//{{V2}}
ORGANIZATION_BLOCK OB1
TITLE= "Cyclic main program"


AUTHOR:nb
FAMILY:nb
NAME:nb
VERSION:1.0


VAR_TEMP
       OB1_EV_CLASS:BYTE //Bits 0-3 = 1 (Coming event), Bits 4-7 = 1 (Event class 1)
       OB1_SCAN_1:BYTE //1 (Cold restart scan 1 of OB 1), 3 (Scan 2-n of OB 1)
       OB1_PRIORITY:BYTE //1 (Priority of 1 is lowest)
       OB1_OB_NUMBR:BYTE //1 (Organization block 1, OB1)
       OB1_RESERVED_1:BYTE //Reserved for system
       OB1_RESERVED_2:BYTE //Reserved for system
       OB1_PREV_CYCLE:INT //Cycle time of previous OB1 scan (milliseconds)
       OB1_MIN_CYCLE:INT //Minimum cycle time of OB1 (milliseconds)
       OB1_MAX_CYCLE:INT //Maximum cycle time of OB1 (milliseconds)
       OB1_DATE_TIME:DATE_AND_TIME //Date and time OB1 started
END_VAR
BEGIN

NETWORK
TITLE=
//{{k}}
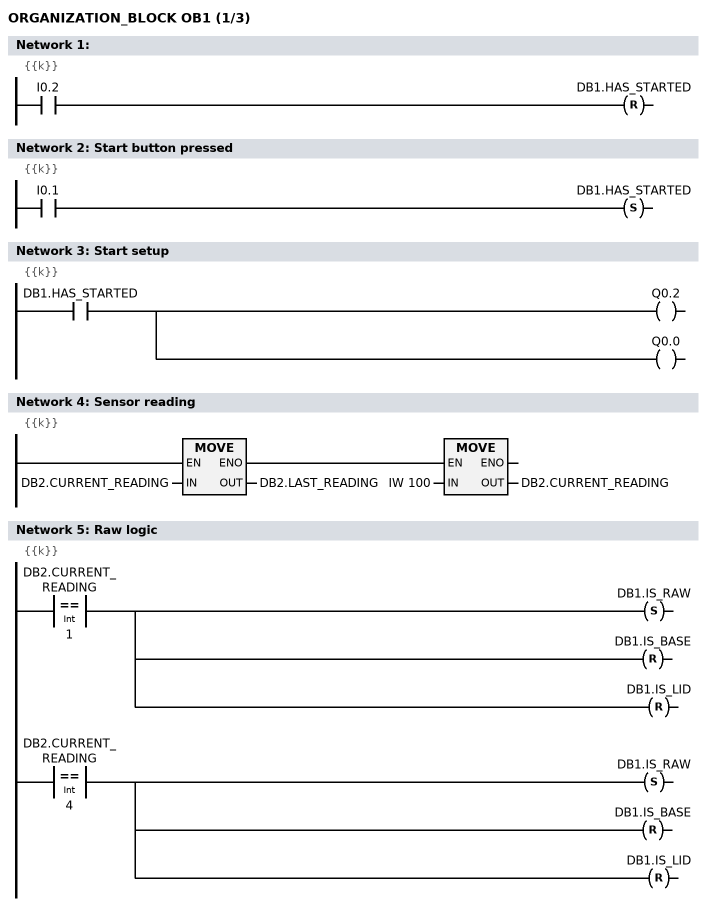

       A    I0.2
       R    DB1.HAS_STARTED

NETWORK
TITLE=Start button pressed
//{{k}}

       A    I0.1
       S    DB1.HAS_STARTED

NETWORK
TITLE=Start setup
//{{k}}

       A    DB1.HAS_STARTED
       =    Q0.2
       =    Q0.0

NETWORK
TITLE=Sensor reading
//{{k}}

       L    DB2.CURRENT_READING
       T    DB2.LAST_READING
       SET
       SAVE
       CLR
       A    BR
       JNB  _001
       L    IW        100
       T    DB2.CURRENT_READING
_001  :NOP  0
NETWORK
TITLE=Raw logic
//{{k}}

       A(
       L    DB2.CURRENT_READING
       L    1
       ==I
       )
       S    DB1.IS_RAW
       R    DB1.IS_BASE
       R    DB1.IS_LID
       A(
       L    DB2.CURRENT_READING
       L    4
       ==I
       )
       S    DB1.IS_RAW
       R    DB1.IS_BASE
       R    DB1.IS_LID
NETWORK
TITLE=Raw logic
//{{k}}
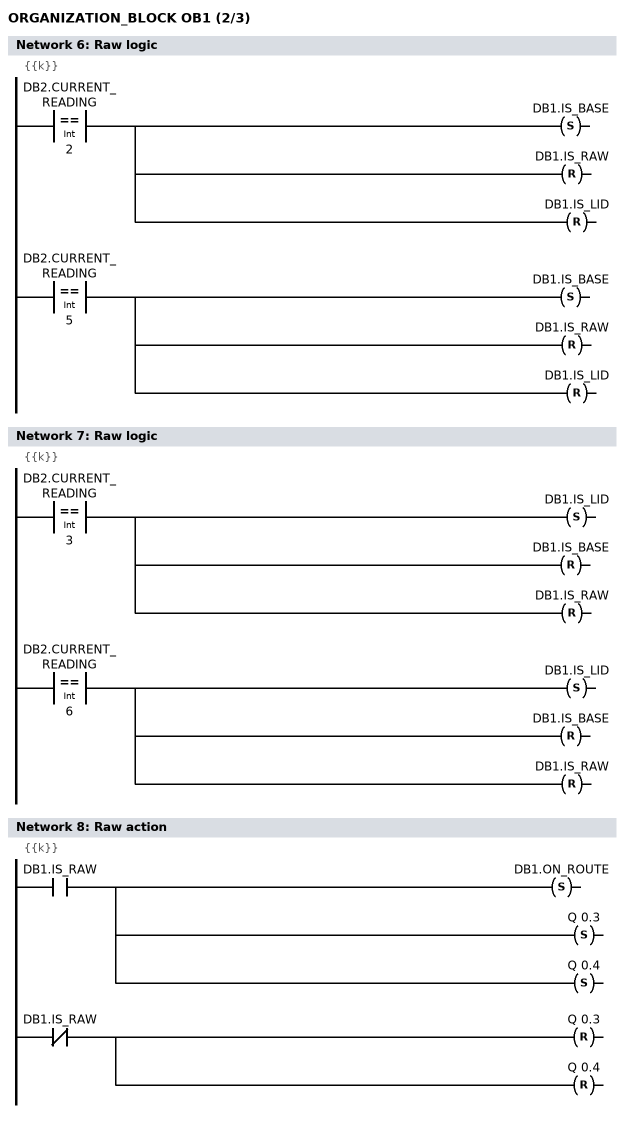

       A(
       L    DB2.CURRENT_READING
       L    2
       ==I
       )
       S    DB1.IS_BASE
       R    DB1.IS_RAW
       R    DB1.IS_LID
       A(
       L    DB2.CURRENT_READING
       L    5
       ==I
       )
       S    DB1.IS_BASE
       R    DB1.IS_RAW

       R    DB1.IS_LID
NETWORK
TITLE=Raw logic
//{{k}}

       A(
       L    DB2.CURRENT_READING
       L    3
       ==I
       )
       S    DB1.IS_LID
       R    DB1.IS_BASE
       R    DB1.IS_RAW

       A(
       L    DB2.CURRENT_READING
       L    6
       ==I
       )
       S    DB1.IS_LID
       R    DB1.IS_BASE
       R    DB1.IS_RAW
NETWORK
TITLE=Raw action
//{{k}}

       A    DB1.IS_RAW
       S    DB1.ON_ROUTE
       S    Q         0.3
       S    Q         0.4
       AN   DB1.IS_RAW
       R    Q         0.3
       R    Q         0.4
NETWORK
TITLE=Base action
//{{k}}
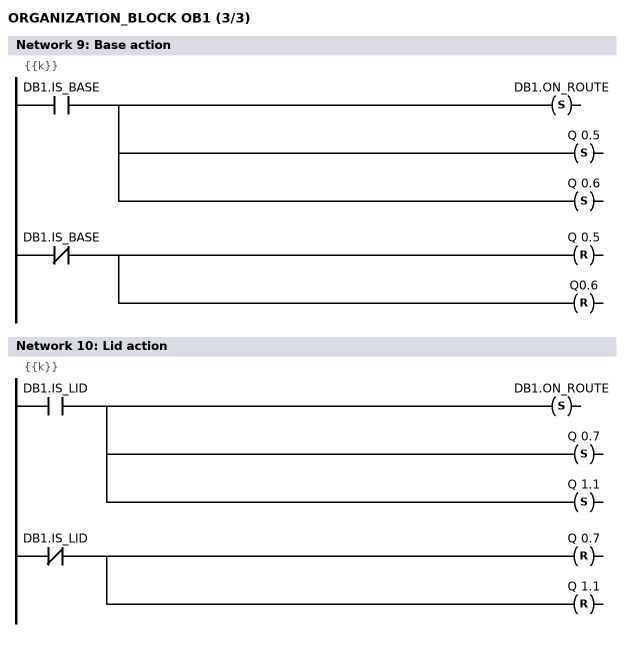

       A    DB1.IS_BASE
       S    DB1.ON_ROUTE
       S    Q         0.5
       S    Q         0.6
       AN   DB1.IS_BASE
       R    Q         0.5
       R    Q0.6
NETWORK
TITLE=Lid action
//{{k}}

       A    DB1.IS_LID
       S    DB1.ON_ROUTE
       S    Q         0.7
       S    Q         1.1
       AN   DB1.IS_LID
       R    Q         0.7
       R    Q         1.1
NETWORK
TITLE=
//{{k}}

       A(
       L    DB2.CURRENT_READING
       L ???
       ==I
       )
END_ORGANIZATION_BLOCK
